(* PLC project Generated.project, CODESYS CODESYS V3.5 SP19 Patch 1 *)
(* stored: creationDateTime 2026-09-19T14:15:31.941995, modificationDateTime 2026-09-19T14:15:31.941995 *)

(* ═══════════════════════════════════════════════════════════════ ⚙️ ST_fbWinchCmdArbitration_Cfg — Config treuil (partagé M1/M2) ─────────────────────────────────────────────────────────────── 🎯 Rôle : Config statique de FB_WinchCmdArbitrationM1/M2. Structure UNIQUE partagée : M1 consomme BtnStepTgt (boutons/both), M2 consomme BtnStepTgt (boutons/both) + plafonds benne par sens. 📤 Producteur : PRG_04_Treuils_Benne (câblage). 📄 Doc : DOC/AF/AF_Partie-10_Fonction_Winch_v2.1.md 🔌 Remplace les paliers codés en dur (StepTgt := 5 / StepTgt := 1) par des constantes nommées. ═══════════════════════════════════════════════════════════════ *)
TYPE ST_fbWinchCmdArbitration_Cfg : STRUCT
  BtnStepTgt : INT := 5;  (* --> [CFG] Palier boutons/both (100 % → palier max) *)
  BucketOverrideStepUpTgt : INT := 1;  (* --> [CFG] Plafond benne montée/fermeture *)
  BucketOverrideStepDownTgt : INT := 1;  (* --> [CFG] Plafond benne descente/ouverture *)
  BucketAutoMaxStepUp : INT := 1;  (* --> [CFG] Plafond AX10 fermeture auto (P1..P2, M2 seul) *)
END_STRUCT;
END_TYPE
